PROGRAM TrafficManager
VAR
	FirstAndMain 	:Intersection;
	SecondAndMain 	:Intersection;
	FirstAndPine	:Intersection;
	SecondAndPine	:Intersection;
	CarSpawner		:TON;
END_VAR

METHOD Init : BOOL
VAR_INPUT
	First, Second, Main, Pine :TrafficDensity;
END_VAR
FirstAndMain.Change_TrafficFlow(TrafficDensity.Low,TrafficDensity.Medium, North, West);
SecondAndMain.Change_TrafficFlow(TrafficDensity.Medium,TrafficDensity.Medium, North, East);

FirstAndPine.Change_TrafficFlow(TrafficDensity.Low,TrafficDensity.High, South, West);
SecondAndPine.Change_TrafficFlow(TrafficDensity.Medium,TrafficDensity.High, South, East);
END_METHOD

METHOD Update
VAR_INPUT
END_VAR
FirstAndMain.UpdateLights();
SecondAndMain.UpdateLights();
//			  |						   |
//---------------<-Main Street->------------------
//		First |					Second |
//			  |						   |
//			  |  					   |
//----------------<-Pine Street->------------------
//			  |						   |
FirstAndPine.UpdateLights();
SecondAndPine.UpdateLights();


UpdateCars();
END_METHOD

METHOD UpdateCars : BOOL
VAR_INPUT
END_VAR
CarSpawner(IN := NOT CarSpawner.Q, PT := T#1S);
IF CarSpawner.Q THEN
	FirstAndMain.CarQueue;
	SecondAndMain.CarQueue;
	FirstAndPine.CarQueue;
	SecondAndPine.CarQueue;
END_IF
END_METHOD

END_PROGRAM

(* stored: Version 1.1.0.1, ProductVersion 3.1.4024.11
   POU TrafficManager: Id {f9cd464c-baa3-4ab8-8ab5-576788caeb1f}, SpecialFunc None
   Method Init: Id {4af402df-6d40-4d47-9111-d375f8a9ea95}
   Method Update: Id {8e35d2c6-934a-4647-9bfc-9e09ec83a63a}
   Method UpdateCars: Id {892be0b6-8b1a-4845-81d2-2c82026e0563} *)
